FUNCTION_BLOCK FB_HMI_CABINETS EXTENDS FB_HMI_COMPONENT
VAR_INPUT
END_VAR
VAR_OUTPUT
END_VAR
VAR
END_VAR

END_FUNCTION_BLOCK

(* stored: Version 1.1.0.1, ProductVersion 3.1.4024.14
   POU FB_HMI_CABINETS: Id {7cfce7ac-44b3-4d04-a8cd-813baf72c575}, SpecialFunc None *)
